# EPICS alarm handler configuration: mps_database/bare/alarms/areas/mpln_bpn14_mp01.alhConfig
GROUP NULL MPLN:BPN14:MP01:1
$ALIAS MPS Link Node 78
$GUIDANCE
LTUH MPS
   Group Name: MPLN:BPN14:MP01:1
   Summary PV:  MPLN:BPN14:MP01:1:STATSUMY
$END
CHANNEL  MPLN:BPN14:MP01:1    MPLN:BPN14:MP01:1:MPS_EN_RBV		-----
CHANNEL  MPLN:BPN14:MP01:1    MPLN:BPN14:MP01:1:LC1_MODE_RBV		-----
